{attribute addProperty BoxType "EL6002-0000-0017"}
{attribute addProperty Id "COM_TxPDO_Map_Inputs_ChannelAT %I*ARRAY[0..1] OF COM_TxPDO_Map_Inputs_Channel_85D1D733384480COM_RxPDO_Map_Outputs_ChannelAT %Q*ARRAY[0..1] OF COM_RxPDO_Map_Outputs_Channel_85BCA431384480WcStateAT %I*WcState_F855686C1620InfoDataAT %I*InfoData_BC63D37F80100"}
{attribute addProperty CRC "749490506"}
{attribute addProperty SizeInBites "864"}
{attribute addProperty SizeInBytes "108"}
TYPE EL6002_45B1C254 :
STRUCT
	{attribute addProperty Name "COM_TxPDO_Map_Inputs_Channel"}
	COM_TxPDO_Map_Inputs_Channel : ARRAY[0..1] OF COM_TxPDO_Map_Inputs_Channel_85D1D733;
	{attribute addProperty Name "COM_RxPDO_Map_Outputs_Channel"}
	COM_RxPDO_Map_Outputs_Channel : ARRAY[0..1] OF COM_RxPDO_Map_Outputs_Channel_85BCA431;
	{attribute addProperty Name "WcState"}
	WcState : WcState_F855686C;
	{attribute addProperty Name "InfoData"}
	InfoData : InfoData_BC63D37F;
END_STRUCT
END_TYPE

(* stored: Version 1.2.0.0, ProductVersion 3.1.4024.9
   DUT EL6002_45B1C254: Id {615ba57a-6f18-4e00-a320-394620ba6505} *)
